// SIMATIC S7-200 project (STEP 7-Micro/WIN), CPU 221 REL 01.10

ORGANIZATION_BLOCK 主程序:OB1
TITLE=程序注释
BEGIN
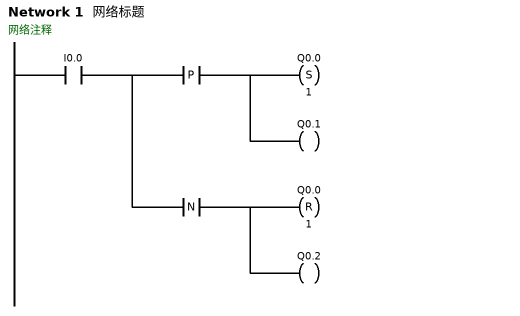
Network 1 // 网络标题
// 网络注释
LD     I0.0
LPS
EU
S      Q0.0, 1
=      Q0.1
LPP
ED
R      Q0.0, 1
=      Q0.2
END_ORGANIZATION_BLOCK
